Universal Robots PolyScope program: taskboard_bearing_turn_right.urp

Program taskboard_bearing_turn_right (installation=default directory=/programs/wrs2020 createdIn=5.7.0.90932 lastSavedIn=5.10.0.106288 robotSerialNumber=20205500607)
Calibrated DH parameters: a=[0.000096, -0.337, -0.383372, 0.000118, 0.000015, 0]; d=[0.162724, 79.377998, -95.545185, 16.300583, 0.099689, 0.099499]; alpha=[1.569249, 0.003272, 0.005201, 1.570041, -1.570219, 0]; deltaTheta=[0, 0.65664, 5.410619, 0.215927, -0.000001, 0]
Robot Program (runOnlyOnce=true)
  URCap Gripper (Robotiq_Grippers, Robotiq Inc.) dataModel(position=0.0, force=0.0, speed=100.0, positionInDouble=0.0, forceInDouble=0.0, speedInDouble=100.0, slaveIds=[9], blocking=true)
  MoveJ speed 60 deg/s, acceleration 80 deg/s^2 (useActiveTCP=false) tcp=gripper_85_tip; feature=Base
    Waypoint athole: TCP in base x=-103.244 y=-570.103 z=229.07 mm, rx=1.4967 ry=-1.6177 rz=-0.8284 rad; joints [89.403, -71.985, 105.307, -128.547, -149.863, -89.084] deg; TCP offset x=0 y=0 z=165 mm, rx=0 ry=0 rz=0 rad
    'At taskboard bearing'
  URCap Gripper (Robotiq_Grippers, Robotiq Inc.) dataModel(position=100.0, force=100.0, speed=100.0, positionInDouble=100.0, forceInDouble=100.0, speedInDouble=100.0, slaveIds=[9], blocking=true)
  Force Frame feature=Base; selection=[1, 0, 0, 0, 0, 0]; wrench=[-10, 0, 10, 0, 0, 0]; limitsForce=[0.01, 0.15, 0.01, 1.047198, 1.047198, 1.047198]; limitsMotion=[0.1, 0.1, 0.1, 0.349066, 0.349066, 0.349066]
    MoveL speed 50 mm/s, acceleration 200 mm/s^2 (useActiveTCP=false) tcp=gripper_85_tip; feature=Base
      Waypoint rightturn_small (Relative): relativeFromPosition TCP in base x=-93.069 y=-570.049 z=228.937 mm, rx=1.497 ry=-1.6176 rz=-0.8285 rad; joints [90.445, -71.969, 104.759, -126.217, -149.936, -87.029] deg; TCP in base x=-103.09 y=-571.303 z=229.127 mm, rx=1.4379 ry=-1.625 rz=-0.735 rad; joints [89.37, -72.375, 108.099, -137.424, -149.699, -90.269] deg
      SuppressedNode
        Waypoint rightturn (Relative): relativeFromPosition TCP in base x=-93.069 y=-570.049 z=228.937 mm, rx=1.497 ry=-1.6176 rz=-0.8285 rad; joints [90.445, -71.969, 104.759, -126.217, -149.936, -87.029] deg; TCP in base x=-93.056 y=-570.054 z=228.975 mm, rx=1.1857 ry=-1.6671 rz=-0.4357 rad; joints [90.457, -71.686, 115.038, -161.493, -150.211, -86.762] deg
      SuppressedNode
        Waypoint leftturn_small (Relative): relativeFromPosition TCP in base x=-93.048 y=-570.049 z=228.934 mm, rx=1.1858 ry=-1.6671 rz=-0.4357 rad; joints [90.457, -71.685, 115.04, -161.493, -150.208, -86.762] deg; TCP in base x=-102.652 y=-571.796 z=229.176 mm, rx=1.2628 ry=-1.6509 rz=-0.5062 rad; joints [89.296, -72.027, 113.875, -158.069, -149.327, -90.488] deg
      SuppressedNode
        Waypoint leftturn (Relative): relativeFromPosition TCP in base x=-93.048 y=-570.049 z=228.934 mm, rx=1.1858 ry=-1.6671 rz=-0.4357 rad; joints [90.457, -71.685, 115.04, -161.493, -150.208, -86.762] deg; TCP in base x=-93.069 y=-570.047 z=228.952 mm, rx=1.497 ry=-1.6176 rz=-0.8285 rad; joints [90.445, -71.97, 104.758, -126.214, -149.936, -87.03] deg
  URCap Gripper (Robotiq_Grippers, Robotiq Inc.) dataModel(position=0.0, force=0.0, speed=100.0, positionInDouble=0.0, forceInDouble=0.0, speedInDouble=100.0, slaveIds=[9], blocking=true)
  MoveJ speed 60 deg/s, acceleration 80 deg/s^2 (useActiveTCP=false) tcp=gripper_85_tip; feature=Base
    Waypoint athole: TCP in base x=-103.244 y=-570.103 z=229.07 mm, rx=1.4967 ry=-1.6177 rz=-0.8284 rad; joints [89.403, -71.985, 105.307, -128.547, -149.863, -89.084] deg
